// TwinCAT 3 PLC project Project1_1
// ProgramVersion: 3.1.4020.2
// libraries:
//   Tc2_Standard, * (Beckhoff Automation GmbH)
//   Tc2_System, * (Beckhoff Automation GmbH)
//   Tc3_Module, * (Beckhoff Automation GmbH)
// project tree:
//   / GlobalTextList.TcGTLO, PlcTask.TcTTO, Visualization Manager.TcVMO (not stored)
//   POUs/ MAIN.TcPOU
//   VISUs/ Visualization_1.TcVIS

CONFIGURATION Project1_1
    RESOURCE PLC ON TwinCAT3
        TASK PlcTask(INTERVAL := T#10ms, PRIORITY := 20);
        PROGRAM MAIN WITH PlcTask : MAIN;
    END_RESOURCE
END_CONFIGURATION

// ---- POUs/MAIN.TcPOU
PROGRAM MAIN
VAR

// Outputs
Motor : BOOL;
Valve : BOOL;
Tank_empty_out : BOOL;

// Inputs
Container_in_place : BOOL;
Container_full : BOOL; 
Tank_empty_in : BOOL;  
Loading : BOOL; 
Unloading : BOOL; 
START : BOOL; 
STOP : BOOL; 
EMERGENCY : BOOL;
Refill : BOOL;	// Input that represents the tank's refill

// Internal Variables
Count : INT;	// Variable that represent the number of containers that the system processed
State: INT;		// Variable that represent the number of the state of the system's process
S1 : BOOL;		// Variable that is TRUE after loading is TRUE, meaning that the container is carried to the tank
S2 : BOOL;		// Variable that is TRUE after container in place is TRUE, meaning that the container is being fill by the tank
S3 : BOOL;		// Variable that is TRUE after container full is TRUR, meaning that the container is carried to the unloading point
RESET : BOOL;	// Variable that is TRUE when TANK EMPTY pass from TRUE TO FALSE.

END_VAR

// IMPLEMENTATION ------------------------------------------------------------------------------

// When EMERGENCY button is pressed, the motor and valve stop and the system does nothing
IF EMERGENCY = TRUE THEN
	MOTOR:=FALSE;
	VALVE:=FALSE;
ELSE
	// If the EMERGENCY button is OFF, the system check what is the state that he was before EMERGENCY, and continue the process
	CASE State OF
		
		// If the system is in the State 0, he should wait for the START button to be pressed. If the tank is empty, the system should continue is this state, ignoring the START button.
		// TANK_EMPTY_IN is normally pressed contact in such a way that it outputs FALSE when sensing water and TRUE when the tank is empty.
		0: IF TANK_EMPTY_IN = TRUE THEN			
			RESET := TRUE;
			START := FALSE;
		END_IF
		TANK_EMPTY_OUT := TANK_EMPTY_IN;
		IF REFILL =TRUE THEN
			TANK_EMPTY_OUT := FALSE;
			TANK_EMPTY_IN := FALSE;
		END_IF
		// Every time that the tank is not empty, the system should reset the counter. In other words, if the tank was empty and it is now full, it means that he has capacity for 10 new containers.
		IF START AND NOT TANK_EMPTY_IN = TRUE THEN
			IF RESET =TRUE THEN
				COUNT :=0;
				RESET := FALSE;
			END_IF
			State:= State+1;	// If the condition of changing the state is fulfilled, the State variable should increment 1 for the system to jump to the next state
		END_IF
		
		// If the system is in the State 1, he should wait for the LOADING button to be pressed. If the user click on STOP button or if, for some reason, the tank is empty, the system should go to the State 0.
		1: IF TANK_EMPTY_IN =TRUE  OR STOP =TRUE THEN
			State := 0;
			START := FALSE;
		END_IF 
		// If the LOADING button is pressed, the motor starts to run and we increment 1 to the State variable to jump to the next State
		IF Loading = TRUE THEN
			MOTOR := TRUE;
			State:= State+1 ;
			S1 := TRUE; 
		END_IF
		
		// If the system is in the State 2, he should wait for the CONTAINER_IN_PLACE button to be pressed.
		2: MOTOR:=TRUE;
		// If that button is pressed, the motor should stop, and the valve must be opened. After that, the state variable should be incremented.
		IF CONTAINER_IN_PLACE = TRUE THEN
			MOTOR:= FALSE;
			S1 :=FALSE;
			S2 := TRUE;
			State:= State+1 ; 
			VALVE:= TRUE;
		END_IF
		
		// If the system is in the State 3, he should wait for the CONTAINER_FULL button to be pressed.
		3: VALVE:=TRUE;
		// If that button is pressed, the motor should be ON and the valve closed. If this happens, the counter should increment 1, meaning that the number of filled containers increased
		IF CONTAINER_FULL = TRUE THEN
			COUNT := COUNT+1; 
			VALVE:= FALSE ;
			S2 := FALSE;
			S3:=TRUE;
			CONTAINER_FULL := FALSE;
			CONTAINER_IN_PLACE := FALSE;
			MOTOR:= TRUE ; 
			State:= State+1 ; 
		END_IF
		
		// If the system is in the State 4, he shoul wait for the UNLOADING button to be pressed
		4:  MOTOR:=TRUE;
		// If the UNLOADING button is pressed, the system have to check if the counter is bigger or equal than 10 OR if the STOP button was pressed. In that case, the system should go to State 0
		IF (UNLOADING AND (COUNT >10 OR COUNT = 10)) OR (UNLOADING AND STOP) THEN
			IF (UNLOADING AND (COUNT >10 OR COUNT = 10)) THEN
				TANK_EMPTY_OUT := TRUE;
				TANK_EMPTY_IN := TRUE ;
			END_IF
			MOTOR := FALSE;
			STATE := 0; 
			S3:=FALSE;
		ELSE 
		// If the UNLOADING button was pressed and the counter was lower than 10 or if the STOP button was not pressed, he should go to the State 1 and wait for another container to fill
		IF  UNLOADING AND COUNT < 10 THEN
			MOTOR := FALSE;
			STATE := 1;
			S3:=FALSE;
			END_IF	
		END_IF
	END_CASE
	
END_IF

END_PROGRAM

// ---- GlobalTextList.TcGTLO
TEXTLIST GlobalTextList
  1 = 'Container full'
  0 = 'Container in place'
  7 = 'Emergency'
  3 = 'Loading'
  8 = 'Motor'
  11 = 'Not Running'
  13 = 'Refiil tank'
  14 = 'Refill tank'
  10 = 'Running'
  5 = 'Start'
  6 = 'Stop'
  2 = 'Tank empty'
  12 = 'Tank refill'
  4 = 'Unloading'
  9 = 'Valve'
END_TEXTLIST

// ---- VISUs/Visualization_1.TcVIS
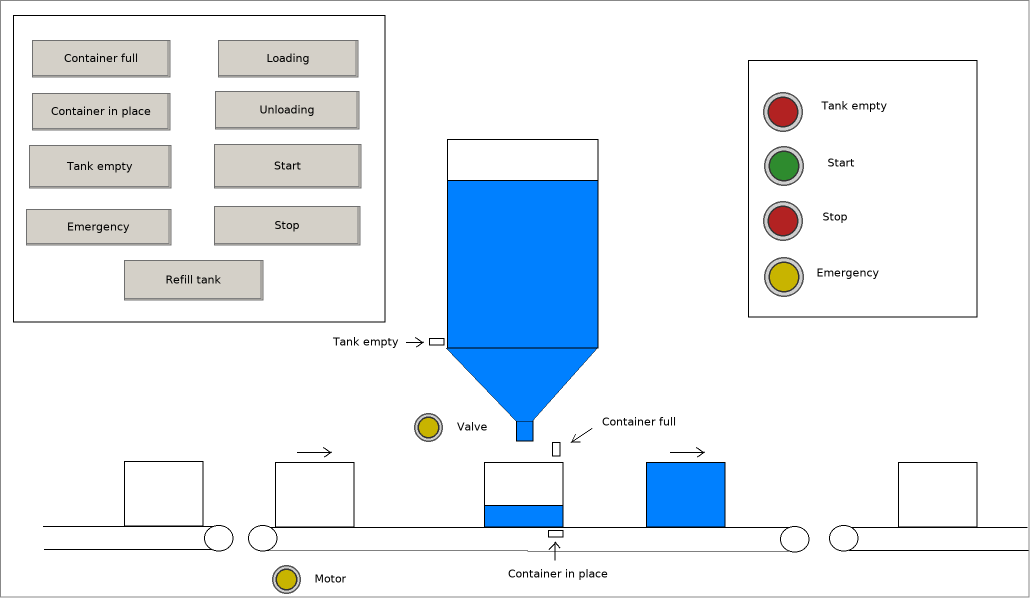
VISUALIZATION Visualization_1  // 1030x598
    Rectangle (13,15 372x307)
    Rectangle (748,60 229x257)
    Button (32,93 138x37), "Container in place", colour toggle: MAIN.Container_in_place
        toggle MAIN.Container_in_place
    Button (32,40 138x37), "Container full", colour toggle: MAIN.Container_full
        toggle MAIN.Container_full
    Button (29,145 142x43), "Tank empty", colour toggle: MAIN.Tank_empty_in
        toggle MAIN.Tank_empty_in
    Button (218,40 140x37), "Loading"
        tap MAIN.Loading
    Button (215,91 144x38), "Unloading"
        tap MAIN.Unloading
    Button (214,144 147x44), "Start", colour toggle: MAIN.Start
        toggle MAIN.Start
    Button (214,206 146x39), "Stop", colour toggle: MAIN.Stop
        toggle MAIN.Stop
    Button (26,209 145x36), "Emergency", colour toggle: MAIN.Emergency
        toggle MAIN.Emergency
    Line (43,526) (222,526)
    Line (44,549) (223,549)
    Ellipse (204,525 29x26)
    Line (256,527) (795,527)
    Line (258,550) (797,551)
    Ellipse (780,526 29x26)
    Ellipse (248,525 29x26)
    Line (848,527) (1027,527)
    Line (849,550) (1028,550)
    Ellipse (829,525 29x26)
    Rectangle (124,461 79x65)
    Rectangle (275,462 79x65), invisible if: NOT MAIN.S1
    Rectangle (484,462 79x65), invisible if: NOT MAIN.S2
    Rectangle (646,462 79x65), invisible if: NOT MAIN.S3
    Rectangle (898,462 79x65)
    Rectangle (447,139 151x209)
    Rectangle (516,420 17x21)
    Line (297,452) (331,452), invisible if: (NOT MAIN.S1) OR (MAIN.EMERGENCY)
    Line (323,447) (330,452), invisible if: (NOT MAIN.S1) OR (MAIN.EMERGENCY)
    Line (331,452) (324,457), invisible if: (NOT MAIN.S1) OR (MAIN.EMERGENCY)
    Line (670,452) (704,452), invisible if: (NOT MAIN.S3) OR (MAIN.EMERGENCY)
    Line (696,447) (703,452), invisible if: (NOT MAIN.S3) OR (MAIN.EMERGENCY)
    Line (704,452) (697,457), invisible if: (NOT MAIN.S3) OR (MAIN.EMERGENCY)
    Line (406,342) (423,342)
    Line (415,337) (422,342)
    Line (423,342) (416,347)
    Line (555,560) (555,542)
    Line (549,549) (555,543)
    Line (560,548) (555,542)
    Rectangle (429,338 15x7)
    Rectangle (548,530 15x7)
    Rectangle (552,442 8x14)
    Line (571,442) (592,428)
    Line (575,434) (571,442)
    Line (580,442) (572,442)
    Lamp1 (760,84 46x56), variable: MAIN.Tank_empty_out, style: Lamp-Lamp1-Red
    Label (812,91 85x30), "Tank empty"
    Lamp1 (761,138 46x56), variable: MAIN.Start, style: Lamp-Lamp1-Green
    Lamp1 (760,193 46x56), variable: MAIN.Stop, style: Lamp-Lamp1-Red
    Label (481,552 154x44), "Container in place"
    Label (289,320 154x44), "Tank empty"
    Label (562,400 154x44), "Container full"
    Rectangle (447,180 151x168), invisible if: MAIN.Tank_empty_in
    Rectangle (516,420 17x21), invisible if: MAIN.Tank_empty_in
    Rectangle (484,505 79x22), invisible if: NOT MAIN.S2
    Label (817,148 48x30), "Start"
    Label (809,202 52x30), "Stop"
    Lamp1 (270,563 33x33), variable: MAIN.Motor, style: Lamp-Lamp1-Yellow
    Label (303,564 55x30), "Motor"
    Lamp1 (412,411 33x33), variable: MAIN.Valve, style: Lamp-Lamp1-Yellow
    Label (445,412 55x30), "Valve"
    Lamp1 (761,249 46x56), variable: MAIN.Emergency, style: Lamp-Lamp1-Yellow
    Label (807,258 82x30), "Emergency"
    Button (124,260 139x40), "Refill tank"
        tap MAIN.Refill
    Polygon (446,348) (523,348) (597,348) (532,421) (516,421), colour toggle: MAIN.Tank_empty_in
END_VISUALIZATION
